(* CODESYS project xlh_control_systems_00_10.library
   Author: Pascal Helfenstein - Thomas Ruoss
   Version: 0.1
   Title: xLH Control Systems
   DefaultNamespace: XlhControlSystems
   Placeholder: XlhControlSystems
   Company: xemax ag

Project tree, tasks and I/O mapping:
  libraries: Standard, 3.5.22.0 (System); VisuDialogs, * (System)
  00000000-0000-0000-0000-000000000000|D:\CoDeSys\LibrariesV3\trunk\Intern\CAA\CAA Template\3.2.0.3 draft\Prefix.pdf
  00000000-0000-0000-0000-000000000000|D:\CoDeSys\LibrariesV3\trunk\Intern\CAA\CAA Template\3.4.0.0 draft\Placeholder.xml
  00000000-0000-0000-0000-000000000000|D:\CoDeSys\LibrariesV3\trunk\Intern\CAA\CAA Template\3.5.2.0 draft\Placeholder.xml
  Library Information/
    function GetLibVersion [ST]
    function GetLibVersionNumber [ST]
    function IsLibReleased [ST]
  POUs/
    function block DT1 [ST]: reset
    data type eFilterType
    data type eControllerType
    data type eSignalShape
    function block I [ST]
    function block CharacteristicCurve [ST]
    function block Limitation [ST]
    function block Deadband [ST]
    function block Logger_ [ST]
    function block P [ST]
    function block PT1 [ST]: reset
    function block PT2 [ST]: reset
    function block PT2s [ST]: reset
    function block PTt [ST]: reset
    function block SignalNoise [ST]
    function block Controller [ST]: controllerType, reset
    program CS_COMMOM [ST]
    function block SignalGenerator [ST]
    text list GlobalTextList
    TOOLBOX/
      function block KalmanFilter [ST]: reset
      function LrealToInt [ST]
      function LrealToUInt [ST]
  visualisation CS_VISU_SignalGenerator
  visualisation CS_VISU_DT1
  visualisation CS_VISU_SignalNoise
  visualisation VISU_HELPER_Combobox_eSignalShape
  visualisation CS_VISU_P
  visualisation CS_VISU_KalmanFilter
  text list TextListForCombobox_eSignalShape
  visualisation CS_VISU_CharacteristicCurve
  visualisation CS_VISU_PTt
  visualisation CS_VISU_Limitation
  visualisation CS_VISU_I
  visualisation CS_VISU_PT1
  visualisation CS_VISU_Controller
  visualisation CS_VISU_PT2
  visualisation VISU_HELPER_Combobox_eControllerType
  visualisation CS_VISU_PT2s
  visualisation CS_VISU_Deadband
  text list TextListForCombobox_eControllerType
  program README [ST]
*)

// POUs/eFilterType
(*
eFilterType — Selects the filter type.
*)
TYPE eFilterType :
(
	NONE_ := 1,     // No filtering
	LOW_PASS := 2,  // Low-pass filter
	HOCH_PASS := 3  // High-pass filter (German identifier "Hochpass" kept for backward compatibility)
)INT;
END_TYPE

// POUs/eControllerType
(*
eControllerType — Selects the controller structure used by the Controller function block.
*)
TYPE eControllerType :
(
	P := 1,     // Proportional controller
	I := 2,     // Integral controller
	PI := 3,    // Proportional-integral controller
	PDT1 := 4,  // Proportional-derivative controller (D-part with first-order lag)
	PIDT1 := 5  // Proportional-integral-derivative controller (D-part with first-order lag)
)INT;
END_TYPE

// POUs/eSignalShape
(*
eSignalShape — Selects the output waveform of the SignalGenerator function block.
*)
TYPE eSignalShape :
(
	OFF := 1,       // Generator off, output is 0.0
	OFFSET := 2,    // Constant output value (offset only)
	RECTANGLE := 3, // Square wave
	TRIANGLE := 4,  // Triangle wave
	SINUS := 5,     // Sine wave
	RAMP := 6       // Ramp towards a target value with adjustable slope
)INT;
END_TYPE

// Library Information/GetLibVersion
// This function has been automatically generated from the project information.
FUNCTION GetLibVersion : VERSION
VAR_INPUT
	
END_VAR

GetLibVersion.uiMajor := 0;
GetLibVersion.uiMinor := 1;
GetLibVersion.uiServicePack := 65535;
GetLibVersion.uiPatch := 65535;

END_FUNCTION

// Library Information/GetLibVersionNumber
// This function has been automatically generated from the project information.
FUNCTION GetLibVersionNumber : DWORD
VAR_INPUT
	
END_VAR

GetLibVersionNumber := 131071;

END_FUNCTION

// Library Information/IsLibReleased
// This function has been automatically generated from the project information.
FUNCTION IsLibReleased : BOOL
VAR_INPUT
	
END_VAR

IsLibReleased := FALSE;

END_FUNCTION

// POUs/DT1
(*
DT1 — Derivative element with first-order lag (real differentiator).

Transfer function: G(s) = Tv*s / (1 + Tvz*s)

The block is discretized with the explicit Euler method using the global
cycle time CS_COMMOM.fdt. If fTvz <= 0.0 the internal deltas are not
updated and the output keeps decaying with the last calculated values.
*)
{attribute 'FBVisuCreator'}
{attribute 'FBVisuCreatorPrefix' :=  'CS_VISU_'}
FUNCTION_BLOCK DT1
VAR_INPUT
	{attribute 'FBVisuCreatorFormatString' := '%1.3f'}
	fX: LREAL; // Input signal
	{attribute 'FBVisuCreatorFormatString' := '%1.3f'}
	fTv: LREAL; // Derivative time Tv [s]
	{attribute 'FBVisuCreatorFormatString' := '%1.3f'}
	fTvz: LREAL; // Lag time constant Tvz (T1) [s] of the derivative element
	{attribute 'FBVisuCreatorBoolColor' := 'Red'}
	{attribute 'FBVisuCreatorCustomName' := 'Reset'}
	bReset: BOOL; // TRUE: reset output and internal states to 0.0
END_VAR
VAR_OUTPUT
	{attribute 'FBVisuCreatorFormatString' := '%1.3f'}
	fY: LREAL; // Differentiated output signal
END_VAR
VAR
	fDxe: LREAL; // Output increment caused by the input change
	fDxa: LREAL; // Output decrement caused by the first-order decay
	fEold: LREAL; // Input value of the previous cycle
END_VAR

// Discrete DT1 algorithm: differentiate the input change, output decays with time constant Tvz
IF (fTvz > 0.0) THEN
	fDxe := fTv/fTvz*(fX - fEold);
	fEold := fX;
	fDxa := fY/fTvz*CS_COMMOM.fdt;
END_IF
fY := fY + fDxe - fDxa;

IF bReset THEN
	reset();
END_IF

ACTION reset:
// Reset output and all internal states
fY := 0.0;
fEold := 0.0;
fDxe := 0.0;
fDxa := 0.0;
END_ACTION

END_FUNCTION_BLOCK

// POUs/CS_COMMOM
(*
CS_COMMOM — Common settings of the control system library.

Provides the cycle time fdt that all dynamic function blocks of this
library (PT1, PT2, I, DT1, Controller, SignalGenerator, ...) use for their
discrete-time calculations. fdt must be set to the cycle time of the task
in which those function blocks are called.

Note: the name "COMMOM" (instead of "COMMON") is kept for backward
compatibility with existing applications.
*)
PROGRAM CS_COMMOM
VAR_INPUT
	fdt: LREAL := 0.004; // Cycle time [s] of the calling task
END_VAR

END_PROGRAM

// POUs/PT1
(*
PT1 — First-order lag element (low-pass).

Transfer function: G(s) = K / (1 + T*s)

The block is discretized with the explicit Euler method using the global
cycle time CS_COMMOM.fdt. If fT <= 0.0 the input is passed through directly.
*)
{attribute 'FBVisuCreator'}
{attribute 'FBVisuCreatorPrefix' :=  'CS_VISU_'}
FUNCTION_BLOCK PT1
VAR_INPUT
	{attribute 'FBVisuCreatorFormatString' := '%1.3f'}	
	fX: LREAL; // Input signal
	{attribute 'FBVisuCreatorFormatString' := '%1.3f'}
	fK: LREAL; // Gain K
	{attribute 'FBVisuCreatorFormatString' := '%1.3f'}
	fT: LREAL; // Time constant T [s]
	{attribute 'FBVisuCreatorBoolColor' := 'Red'}
	{attribute 'FBVisuCreatorCustomName' := 'Reset'}
	bReset: BOOL; // TRUE: reset output to 0.0
END_VAR
VAR_OUTPUT
	{attribute 'FBVisuCreatorFormatString' := '%1.3f'}
	fY: LREAL; // Filtered output signal
END_VAR

IF bReset THEN
	reset();
END_IF

// Discrete PT1 algorithm (explicit Euler); pass-through if no time constant is set
IF (fT > 0.0) THEN
	fY := fY + (-fY + fK*fX)/MAX(fT,0.001)*CS_COMMOM.fdt;
ELSE
	fY := fX;
END_IF

ACTION reset:
// Reset output
fY := 0.0;
END_ACTION

END_FUNCTION_BLOCK

// POUs/PT2
(*
PT2 — Second-order lag element, parameterized with two time constants.

Transfer function: G(s) = K / ((1 + T1*s) * (1 + T2*s))

The two time constants T1 and T2 are converted into damping (zeta) and
natural angular frequency (omega), then the same discrete algorithm as in
PT2s is applied using the global cycle time CS_COMMOM.fdt.
*)
{attribute 'FBVisuCreator'}
{attribute 'FBVisuCreatorPrefix' :=  'CS_VISU_'}
FUNCTION_BLOCK PUBLIC PT2
VAR_INPUT
	{attribute 'FBVisuCreatorFormatString' := '%1.3f'}
	fX: LREAL; // Input signal
	{attribute 'FBVisuCreatorFormatString' := '%1.3f'}
	fK: LREAL; // Gain K
	{attribute 'FBVisuCreatorFormatString' := '%1.3f'}
	fT1: LREAL; // First time constant T1 [s]
	{attribute 'FBVisuCreatorFormatString' := '%1.3f'}
	fT2: LREAL; // Second time constant T2 [s]
	{attribute 'FBVisuCreatorBoolColor' := 'Red'}
	{attribute 'FBVisuCreatorCustomName' := 'Reset'}
	bReset: BOOL; // TRUE: reset output and internal states to 0.0
END_VAR
VAR_OUTPUT
	{attribute 'FBVisuCreatorFormatString' := '%1.3f'}
	fY: LREAL; // Filtered output signal
END_VAR
VAR 
	fZeta: LREAL; // Damping ratio, calculated from T1 and T2
	fOmega: LREAL; // Natural angular frequency [rad/s], calculated from T1 and T2
	fXX: LREAL; // Internal state (first integrator)
	fDx: LREAL; // Increment of the internal state per cycle
	fDy: LREAL; // Increment of the output per cycle
END_VAR

// Convert the time constants T1/T2 into the damping/frequency form used by PT2s
fOmega := 1/SQRT(MAX(fT1*fT2, 0.001));
fZeta := fOmega*(fT1+fT2)/2.0;

IF bReset THEN
	reset();
END_IF

// Discrete PT2 algorithm (two coupled integrators, explicit Euler)
fDy := CS_COMMOM.fdt*fOmega*fXX;
fDx := CS_COMMOM.fdt*fOmega*(fK*fX - fY - 2*fZeta*fXX);
fXX := fXX + fDx;
fY := fY + fDy;

ACTION reset:
// Reset output and internal state
fXX := 0.0;
fY := 0.0;
END_ACTION

END_FUNCTION_BLOCK

// POUs/PT2s
(*
PT2s — Second-order lag element, parameterized with damping and natural frequency
(capable of oscillation for zeta < 1).

Transfer function: G(s) = K / (1/omega^2 * s^2 + 2*zeta/omega * s + 1)

The block is discretized as two coupled integrators (explicit Euler) using
the global cycle time CS_COMMOM.fdt.
*)
{attribute 'FBVisuCreator'}
{attribute 'FBVisuCreatorPrefix' :=  'CS_VISU_'}
FUNCTION_BLOCK PUBLIC PT2s
VAR_INPUT
	{attribute 'FBVisuCreatorFormatString' := '%1.3f'}
	fX: LREAL; // Input signal
	{attribute 'FBVisuCreatorFormatString' := '%1.3f'}
	fK: LREAL; // Gain K
	{attribute 'FBVisuCreatorFormatString' := '%1.3f'}
	fZeta: LREAL; // Damping ratio zeta (< 1.0 results in oscillation)
	{attribute 'FBVisuCreatorFormatString' := '%1.3f'}
	fOmega: LREAL; // Natural angular frequency omega [rad/s]
	{attribute 'FBVisuCreatorBoolColor' := 'Red'}
	{attribute 'FBVisuCreatorCustomName' := 'Reset'}
	bReset: BOOL; // TRUE: reset output and internal states to 0.0
END_VAR
VAR_OUTPUT
	{attribute 'FBVisuCreatorFormatString' := '%1.3f'}
	fY: LREAL; // Filtered output signal
END_VAR
VAR 
	fXX: LREAL; // Internal state (first integrator)
	fDx: LREAL; // Increment of the internal state per cycle
	fDy: LREAL; // Increment of the output per cycle
END_VAR

// Discrete PT2 algorithm (two coupled integrators, explicit Euler)
fDy := CS_COMMOM.fdt*fOmega*fXX;
fDx := CS_COMMOM.fdt*fOmega*(fK*fX - fY - 2*fZeta*fXX);
fXX := fXX + fDx;
fY := fY + fDy;

IF bReset THEN
	reset();
END_IF

ACTION reset:
// Reset output and internal state
fXX := 0.0;
fY := 0.0;
END_ACTION

END_FUNCTION_BLOCK

// POUs/I
(*
I — Integral element (integrator).

Transfer function: G(s) = 1 / (Ti*s)

The input is integrated over time using the global cycle time CS_COMMOM.fdt.
If fTi <= 0.0 the integration is stopped and the output holds its value.
*)
{attribute 'FBVisuCreator'}
{attribute 'FBVisuCreatorPrefix' :=  'CS_VISU_'}
FUNCTION_BLOCK I
VAR_INPUT
	{attribute 'FBVisuCreatorFormatString' := '%1.3f'}
	fX: LREAL; // Input signal
	{attribute 'FBVisuCreatorFormatString' := '%1.3f'}
	fTi: LREAL; // Integration time Ti [s]
	{attribute 'FBVisuCreatorBoolColor' := 'Red'}
	bReset: BOOL; // TRUE: reset the integrator to 0.0
END_VAR
VAR_OUTPUT
	fY: LREAL; // Integrated output signal
END_VAR
VAR
	fSum: LREAL; // Integrator accumulator (internal state)
END_VAR

IF (fTi > 0.0) THEN
	fSum := fSum + 1.0/fTi*fX*CS_COMMOM.fdt;
END_IF
IF bReset THEN
	fSum := 0.0;
END_IF
fY := fSum;

END_FUNCTION_BLOCK

// POUs/Controller
(*
Controller — Universal controller (P, I, PI, PDT1, PIDT1) with anti-windup
and feed-forward input.

Basic controller structure (PID-T1 controller):
G(jw) = Kr*[1 + 1/(Tn*jw) + (Tv*jw)/(1 + Tvz*jw)]

The controller type is selected via eTyp (see eControllerType); the action
controllerType enables the P, I and D parts accordingly. The D part is
implemented as a real (lagged) DT1 element by calling the DT1 base block.
The anti-windup implementation corresponds to the behavior of the
simulation software WinFACT BORIS. All discrete-time calculations use the
global cycle time CS_COMMOM.fdt.
*)
{attribute 'FBVisuCreator'}
{attribute 'FBVisuCreatorPrefix' :=  'CS_VISU_'}
FUNCTION_BLOCK PUBLIC Controller
VAR_INPUT
	{attribute 'FBVisuCreatorCustomName' := 'e'}
	{attribute 'FBVisuCreatorFormatString' := '%1.3f'}
	fE: LREAL; // Control error e (setpoint - actual value)
	{attribute 'FBVisuCreatorCustomName' := 'y_FF'}
	{attribute 'FBVisuCreatorFormatString' := '%1.3f'}
	fY_FF: LREAL; // Feed-forward value
	{attribute 'FBVisuCreatorCustomName' := 'Controller type'}
	{attribute 'FBVisuCreatorFormatString' := 'd'}
	eTyp:  eControllerType; // Controller structure (P, I, PI, PDT1, PIDT1)
	{attribute 'FBVisuCreatorBoolColor' := 'Red'}
	{attribute 'FBVisuCreatorCustomName' := 'Reset'}
	bReset: BOOL; // TRUE: reset all controller states to 0.0
	{attribute 'FBVisuCreatorFormatString' := '%1.3f'}
	fKr: LREAL; // Controller gain Kr
	{attribute 'FBVisuCreatorFormatString' := '%1.3f'}
	fTn: LREAL; // Integral (reset) time Tn [s]
	{attribute 'FBVisuCreatorFormatString' := '%1.3f'}
	fTv: LREAL; // Derivative time Tv [s]
	{attribute 'FBVisuCreatorFormatString' := '%1.3f'}
	fTvz: LREAL; // Time constant T1 [s] for the real (lagged) DT1 behavior
	{attribute 'FBVisuCreatorBoolColor' := 'Red'}
	bEnable_AWU: BOOL := TRUE;  // TRUE: anti-windup active
	{attribute 'FBVisuCreatorFormatString' := '%1.3f'}
	fYlim_max: LREAL := 100.0; // Upper anti-windup limit
	{attribute 'FBVisuCreatorFormatString' := '%1.3f'}
	fYlim_min: LREAL := -100.0; // Lower anti-windup limit
END_VAR
VAR_OUTPUT
	{attribute 'FBVisuCreatorFormatString' := '%1.3f'}
	fY: LREAL; // Manipulated variable (controller output)
	{attribute 'FBVisuCreatorFormatString' := '%1.3f'}
	fProportional: LREAL; // Current P part
	{attribute 'FBVisuCreatorFormatString' := '%1.3f'}
	fIntegral: LREAL; // Current I part
	{attribute 'FBVisuCreatorFormatString' := '%1.3f'}
	fDifferential: LREAL; // Current D (DT1) part
	{attribute 'FBVisuCreatorBoolColor' := 'Red'}
	bAct_UL: BOOL := FALSE; // TRUE: output is limited at the upper limit
	{attribute 'FBVisuCreatorBoolColor' := 'Red'}
	bAct_LL: BOOL := FALSE; // TRUE: output is limited at the lower limit
END_VAR
VAR 
	dt1: DT1; // DT1 base element used for the D part

	// Set in the action controllerType depending on the selected controller type
	bEnKr: BOOL; // Enable signal for the P part
	bEnTn: BOOL; // Enable signal for the I part
	bEnTv: BOOL; // Enable signal for the D part
	//
	
	fIntegralCalc: LREAL; // I-part increment of the current cycle
	
	fDy: LREAL;
	fDx: LREAL;
	fXeAlt: LREAL; // Control error of the previous cycle
	fYcalc: LREAL; // Unlimited controller output
	fYcalc_lim: LREAL;
	fKrCalc: LREAL; // Effective gain (1.0 for a pure I-controller)
	fAvoidZero: LREAL := 0.001; // Minimum divisor to avoid division by zero
	tonStartup: TON;
	bResetTvz: BOOL;
	bP_Controller: BOOL; // TRUE: P controller selected
	bI_Controller: BOOL; // TRUE: I controller selected
	bPI_Controller: BOOL; // TRUE: PI controller selected
	bPDT1_Controller: BOOL; // TRUE: PDT1 controller selected
	bPIDT1_Controller: BOOL; // TRUE: PIDT1 controller selected
END_VAR

// Revision history:
// -------------------------------------------------------------------------------------------------------------
// Basic controller structure (PID-T1 controller):
// G(jw) = Kr*[1+1/(Tn*jw)+(Tv*jw/(1+Tvz*jw)]

controllerType();

///////////////////////////////////////////////////////////////////////////////////////////////////////////////
// Calculation of the P part
IF bEnKr THEN // P part active?
	fKrCalc := fKr;
	fProportional := fKrCalc*fE;
ELSE
	fKrCalc := 1.0; // Must be set to 1.0, otherwise the I part of a pure I-controller would not work due to the controller structure.
	fProportional := 0;
END_IF

///////////////////////////////////////////////////////////////////////////////////////////////////////////////
// Calculation of the I part
IF bEnTn THEN // I part active?
	fIntegralCalc := fKrCalc*(fE*CS_COMMOM.fdt)/MAX(fTn,fAvoidZero);
ELSE
	fIntegral := 0;
END_IF

///////////////////////////////////////////////////////////////////////////////////////////////////////////////
// Anti-windup evaluation, modified: 2020-12-01, tr
IF (fIntegral + fY_FF) >= (fYlim_max - fY_FF) AND fE > 0 AND bEnable_AWU THEN // Hold the I part if yI (I part only) is at the upper limit and w > x
	fIntegral := fIntegral;
ELSIF (fIntegral + fY_FF) <= (fYlim_min + fY_FF) AND fE < 0 AND bEnable_AWU THEN // Hold the I part if yI (I part only) is at the lower limit and w < x
	fIntegral := fIntegral;
ELSE
	fIntegral := fIntegral+ fIntegralCalc; // Integrate / accumulate
END_IF

///////////////////////////////////////////////////////////////////////////////////////////////////////////////
// Calculation of the DT1 part, implemented by calling the DT1 base element
IF bEnTv AND (fTvz >= 2.0*CS_COMMOM.fdt) THEN
	dt1(fX:=fKrCalc*fE, fTv:=fTv , fTvz:=fTvz, fY=>fDifferential);
ELSE
	fDifferential := 0;
END_IF

///////////////////////////////////////////////////////////////////////////////////////////////////////////////
// Sum of all three components (P, I and DT1 part).
// The implementation of the limiting (anti-windup) corresponds to the implementation in BORIS, i.e. as long
// as the sum of the two parts (P + I) is outside the limits, the corresponding limit + D part is output as
// the manipulated variable -> see the following lines. Otherwise all three parts (P + I + D)
// are added. Modified: 2020-12-01, tr
IF fProportional + fIntegral + fY_FF >= (fYlim_max - fY_FF) AND bEnable_AWU THEN
	fYcalc := fYlim_max + fDifferential;

ELSIF fProportional + fIntegral + fY_FF <= (fYlim_min + fY_FF) AND bEnable_AWU  THEN
	fYcalc := fYlim_min + fDifferential;

ELSE
	fYcalc := fProportional + fIntegral + fY_FF + fDifferential;
END_IF

///////////////////////////////////////////////////////////////////////////////////////////////////////////////
// Anti-windup: limit the output and set the limit-active flags
IF bEnable_AWU THEN
	IF fYcalc <= fYlim_max AND fYcalc >= fYlim_min THEN
		bAct_UL := FALSE;
		bAct_LL := FALSE;
	ELSIF fYcalc > fYlim_max THEN
			bAct_UL := TRUE;
			bAct_LL := FALSE;
	ELSIF fYcalc < fYlim_min THEN
		bAct_LL := TRUE;
		bAct_UL := FALSE;
	END_IF
	fY := LIMIT(fYlim_min, fYcalc, fYlim_max);
ELSE
	fY := fYcalc;
	bAct_LL := FALSE;
	bAct_UL := FALSE;
END_IF

IF bReset THEN
	this^.reset();
END_IF

ACTION controllerType:
///////////////////////////////////////////////////////////////////////////////////////////////////////////////
// Selection of the available controller configurations
CASE eTyp OF
	 eControllerType.P:
	 	bP_Controller := TRUE;
		bI_Controller := FALSE;
		bPI_Controller := FALSE;
		bPDT1_Controller := FALSE;
		bPIDT1_Controller := FALSE;
		bEnKr := TRUE; // Enable signal for the P part
		bEnTn := FALSE; // Enable signal for the I part
		bEnTv := FALSE; // Enable signal for the D part

	eControllerType.I:
		bP_Controller := FALSE;
		bI_Controller := TRUE;
		bPI_Controller := FALSE;
		bPDT1_Controller := FALSE;
		bPIDT1_Controller := FALSE;
	 	bEnKr := FALSE; // Enable signal for the P part
		bEnTn := TRUE; // Enable signal for the I part
		bEnTv := FALSE; // Enable signal for the D part
		
		
	 eControllerType.PI:
	 	bP_Controller := FALSE;
		bI_Controller := FALSE;
		bPI_Controller := TRUE;
		bPDT1_Controller := FALSE;
		bPIDT1_Controller := FALSE;
	 	bEnKr := TRUE; // Enable signal for the P part
		bEnTn := TRUE; // Enable signal for the I part
		bEnTv := FALSE; // Enable signal for the D part
				
	eControllerType.PDT1:
		bP_Controller := FALSE;
		bI_Controller := FALSE;
		bPI_Controller := FALSE;
		bPDT1_Controller := TRUE;
		bPIDT1_Controller := FALSE;
	 	bEnKr := TRUE; // Enable signal for the P part
		bEnTn := FALSE; // Enable signal for the I part
		bEnTv := TRUE; // Enable signal for the D part
		
	eControllerType.PIDT1:
		bP_Controller := FALSE;
		bI_Controller := FALSE;
		bPI_Controller := FALSE;
		bPDT1_Controller := FALSE;
		bPIDT1_Controller := TRUE;
	 	bEnKr := TRUE; // Enable signal for the P part
		bEnTn := TRUE; // Enable signal for the I part
		bEnTv := TRUE; // Enable signal for the D part
	
END_CASE
END_ACTION

ACTION reset:
// Reset all controller components and the output
fProportional := 0.0;
fIntegral := 0.0;
fDifferential := 0.0;
dt1.reset();
fY := 0.0;
//rTv := 0.0;
fY := 0.0;
END_ACTION

END_FUNCTION_BLOCK

// POUs/P
(*
P — Proportional element.

Transfer function: G(s) = K

The output is the input multiplied by the gain fK.
*)
{attribute 'FBVisuCreator'}
{attribute 'FBVisuCreatorPrefix' :=  'CS_VISU_'}
FUNCTION_BLOCK P
VAR_INPUT
	{attribute 'FBVisuCreatorFormatString' := '%1.3f'}
	fX: LREAL; // Input signal
	{attribute 'FBVisuCreatorFormatString' := '%1.3f'}
	fK: LREAL; // Proportional gain K
	{attribute 'FBVisuCreatorBoolColor' := 'Red'}
	bReset: BOOL; // TRUE: force output to 0.0
END_VAR
VAR_OUTPUT
	fY: LREAL; // Output signal (fX * fK)
END_VAR

fY := fX*fK;
IF bReset THEN
	fY := 0.0;
END_IF

END_FUNCTION_BLOCK

// POUs/SignalGenerator
(*
SignalGenerator — Test signal generator.

Generates a selectable waveform (off, constant offset, square, triangle,
sine or ramp, see eSignalShape) based on the global cycle time
CS_COMMOM.fdt. Optionally, noise from the SignalNoise function block can
be added to the output.

In RAMP mode the output ramps from the current offset towards the target
value fRamp with the slope fdW_dt; when the target is reached it becomes
the new starting point for the next ramp.
*)
{attribute 'FBVisuCreator'}
{attribute 'FBVisuCreatorPrefix' :=  'CS_VISU_'}
FUNCTION_BLOCK SignalGenerator
VAR_INPUT
	{attribute 'FBVisuCreatorCustomName' := 'Type'}
	{attribute 'FBVisuCreatorFormatString' := 'd'}
	eType: eSignalShape := eSignalShape.OFF; // Selected waveform
	{attribute 'FBVisuCreatorCustomName' := 'Offset'}
	{attribute 'FBVisuCreatorFormatString' := '%1.3f'}
	fOffset: LREAL := 0.0; // Constant offset added to the signal
	{attribute 'FBVisuCreatorCustomName' := 'Ramp target'}
	{attribute 'FBVisuCreatorFormatString' := '%1.3f'}
	fRamp: LREAL := 0.0; // Target value of the ramp (RAMP mode)
	{attribute 'FBVisuCreatorCustomName' := 'Ramp slope'}
	{attribute 'FBVisuCreatorFormatString' := '%1.3f'}
	fdW_dt: LREAL := 1.0; // Slope of the ramp, i.e. 1.0 --> 1.0 dW/dt [units/s]
	{attribute 'FBVisuCreatorCustomName' := 'Amplitude'}
	{attribute 'FBVisuCreatorFormatString' := '%1.3f'}
	fAmplitude: LREAL := 1.0; // Amplitude of the periodic signals
	{attribute 'FBVisuCreatorCustomName' := 'Frequency [Hz]'}
	{attribute 'FBVisuCreatorFormatString' := '%1.5f'}
	fFrequency: LREAL := 1.0; // Frequency of the periodic signals [Hz]
	{attribute 'FBVisuCreatorCustomName' := 'Phase shift [°]'}
	{attribute 'FBVisuCreatorFormatString' := '%1.1f'}
	fPhi: LREAL := 0.0; // Phase shift of the periodic signals [°]
	{attribute 'FBVisuCreatorBoolColor' := 'Red'}
	bSignalNoise: BOOL; // TRUE: add noise to the output signal
	{attribute 'FBVisuCreatorFormatString' := '%1.3f'}
	fSignalNoiseAmplification: LREAL; // Gain of the added noise
END_VAR
VAR_OUTPUT
	{attribute 'FBVisuCreatorFormatString' := '%1.3f'}
	fY: LREAL; // Generated output signal
END_VAR
VAR
	fTime: LREAL; // Elapsed time [s], incremented every cycle
	fSum: LREAL; // Accumulated ramp value (RAMP mode)
	signalNoise: SignalNoise := (fAmplification := 1.0); // Noise generator instance
	fYsin: LREAL; // Intermediate value: sine (TRIANGLE mode)
	fYasin: LREAL; // Intermediate value: arcsine of the sine (TRIANGLE mode)
END_VAR
VAR CONSTANT
	fPi: LREAL := 3.141592653589790; // Circle constant pi
END_VAR

fTime := fTime + CS_COMMOM.fdt;

CASE eType OF
	eSignalShape.OFF:
		fY := 0.0;
		fSum := 0.0;
	
	eSignalShape.OFFSET:
		fY := fOffset;
		fRamp := fOffset;
		
	eSignalShape.RAMP:
		// Ramp towards the target value with the configured slope
		IF fY < fRamp THEN
			fSum := fSum + fdW_dt*CS_COMMOM.fdt;
		ELSIF fY > fRamp THEN
			fSum := fSum - fdW_dt*CS_COMMOM.fdt;
		ELSE
			fY := fRamp;
		END_IF
		
		IF fY = fRamp THEN// Target reached: hold the value (anti-windup)
			fY := fRamp;
			fOffset := fRamp; // Set the new starting point for the next ramp
		ELSE
			fY := fOffset + fSum;
		END_IF
			
	eSignalShape.RECTANGLE:
		// Square wave: sign of the sine determines the output level
		fY := SIN(2*fPi*fFrequency*fTime + fPhi*fPi/180.0);
		IF fY >= 0.0 THEN
			fY := fAmplitude;
		ELSIF fY < 0.0 THEN
			fY :=  -fAmplitude;
		END_IF
		fY := LIMIT(-500.0, fY + fOffset, 500.0);
		fRamp := fOffset;

	eSignalShape.TRIANGLE:
		// Triangle wave: arcsine of a sine yields a triangle shape
		fYsin := SIN(2*fPi*fFrequency*fTime + fPhi*fPi/180.0);
		fYasin := 2*ASIN(fYsin)/fPi;
		fY := fAmplitude*fYasin + fOffset;
		
	eSignalShape.SINUS:
		fY := fAmplitude*SIN(2*fPi*fFrequency*fTime + fPhi*fPi/180.0) + fOffset;
		fRamp := fOffset;
		
	ELSE
		eType := eSignalShape.OFF;
END_CASE
// Optionally add noise to the generated signal
IF bSignalNoise AND (eType <> eSignalShape.OFF) THEN
	signalNoise(fAmplification := fSignalNoiseAmplification);
	fY := fY + signalNoise.fY;
END_IF

END_FUNCTION_BLOCK

// POUs/SignalNoise
(*
SignalNoise — Pseudo-random noise generator.

Outputs a pseudo-random noise signal by cycling through an array of 10000
pre-generated random numbers in the range -1.0 <= rnd < 1.0 (one value per
call) and scaling it with fAmplification. The sequence repeats after
10000 calls.
*)
{attribute 'FBVisuCreator'}
{attribute 'FBVisuCreatorPrefix' :=  'CS_VISU_'}
FUNCTION_BLOCK SignalNoise
VAR_INPUT
	{attribute 'FBVisuCreatorFormatString' := '%1.3f'}
	fAmplification: LREAL; // Noise gain factor
END_VAR
VAR_OUTPUT
	{attribute 'FBVisuCreatorFormatString' := '%1.3f'}
	fY: LREAL; // Noise output signal
END_VAR
VAR
	fSum: LREAL; // Unused (kept for compatibility)
	iI: INT := 0; // Index into the random number array, incremented every call
END_VAR
VAR CONSTANT
	// Array of pre-generated random numbers in the range -1.0 <= rnd < 1.0
